// Mitsubishi GX Works2 project: Project 1   PLC: Q03UDV

PROGRAM MAIN
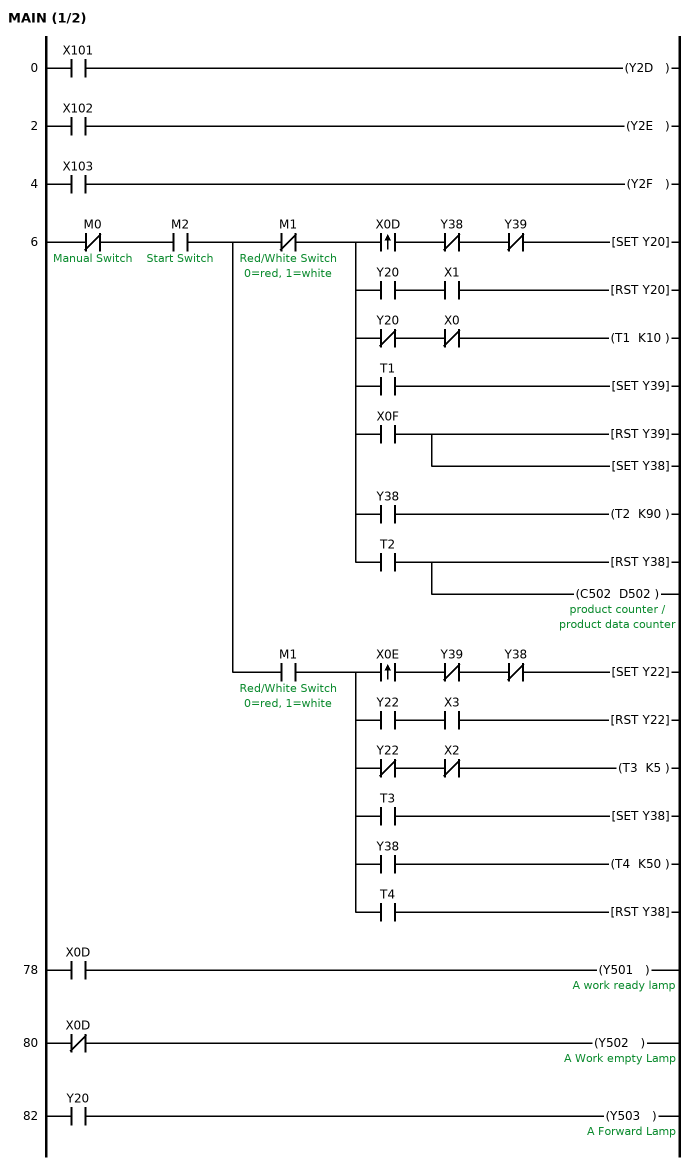
0     LD      X101
      OUT     Y2D
2     LD      X102
      OUT     Y2E
4     LD      X103
      OUT     Y2F
6     LDI     M0  ; Manual Switch
      AND     M2  ; Start Switch
      MPS
      ANI     M1  ; Red/White Switch 0=red, 1=white
      MPS
      ANDP    X0D
      ANI     Y38
      ANI     Y39
      SET     Y20
      MRD
      AND     Y20
      AND     X1
      RST     Y20
      MRD
      ANI     Y20
      ANI     X0
      OUT     T1 K10
      MRD
      AND     T1
      SET     Y39
      MRD
      AND     X0F
      RST     Y39
      SET     Y38
      MRD
      AND     Y38
      OUT     T2 K90
      MPP
      AND     T2
      RST     Y38
      OUT     C502 D502  ; product counter / product data counter
      MPP
      AND     M1  ; Red/White Switch 0=red, 1=white
      MPS
      ANDP    X0E
      ANI     Y39
      ANI     Y38
      SET     Y22
      MRD
      AND     Y22
      AND     X3
      RST     Y22
      MRD
      ANI     Y22
      ANI     X2
      OUT     T3 K5
      MRD
      AND     T3
      SET     Y38
      MRD
      AND     Y38
      OUT     T4 K50
      MPP
      AND     T4
      RST     Y38
78    LD      X0D
      OUT     Y501  ; A work ready lamp
80    LDI     X0D
      OUT     Y502  ; A Work empty Lamp
82    LD      Y20
      OUT     Y503  ; A Forward Lamp
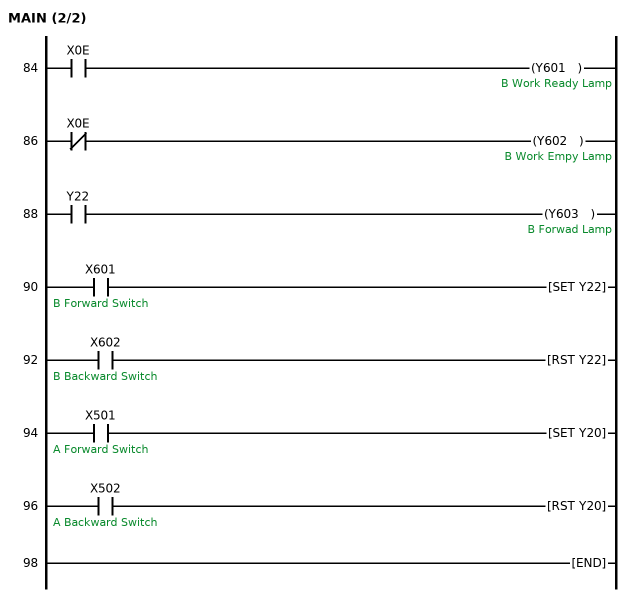
84    LD      X0E
      OUT     Y601  ; B Work Ready Lamp
86    LDI     X0E
      OUT     Y602  ; B Work Empy Lamp
88    LD      Y22
      OUT     Y603  ; B Forwad Lamp
90    LD      X601  ; B Forward Switch
      SET     Y22
92    LD      X602  ; B Backward Switch
      RST     Y22
94    LD      X501  ; A Forward Switch
      SET     Y20
96    LD      X502  ; A Backward Switch
      RST     Y20
98    END
END_PROGRAM

// device comments not shown above
X110  ; A Supply Switch
X120  ; B Supply Switch
X210  ; Motor Forward
X220  ; Motor Backward
X701  ; Conveyor Forward Switch
X702  ; Conveyor Backward Switch
Y802  ; current output
